FUNCTION_BLOCK FB_AxisAbsolute
VAR	
	// =============== Done signals ============================
	_bResetDone			:BOOL;					// Status of function block MC_Reset
	_bHaltDone			:BOOL;					// Status of function block MC_Halt
	_bStopDone			:BOOL;					// Status of function block MC_Stop
	_bMoveDone			:BOOL;					// Status of function block MC_MoveAbsolute

	// =============== State variables ========================
	_bStatusEnable		:BOOL;					// Enable feedback
	_bStateError		:BOOL;					// Error signal
	_bMoveCommandAborted:BOOL;					// Status of function block MC_MoveAbsolute	
	_nStateErrorID		:UDINT;					// Error ID
	_bStateMoving		:BOOL;					// Status of moving
	_fStateActPos		:LREAL;					// Actual Position
	
	// =============== Position Velocity, override ============
	_fTargetPosition	:LREAL;					// Target Position 
	_fTargetVelocity	:LREAL;					// Target Velocity
	fOverride 			:LREAL := 100.0;		// Override 100%
	
	// =============== Axis Limit =============================
	_fMaxPosition		:LREAL;					//	MAX Target Position 
	_fMinPosition		:LREAL;					//	MIN Target Position 
	_fMaxVelocity		:LREAL;					//	MAX Target Velocity
	_fMinVelocity		:LREAL;					//	MIN Target Velocity
	
	// =============== Trigger function blocks ================
	fbTriggerReset		:R_TRIG;				// Trigger to recognize rising edge of reset input
	fbTriggerHalt		:R_TRIG;				// Trigger to recognize rising edge of halt input
	fbTriggerStop		:R_TRIG;				// Trigger to recognize rising edge of stop input
	fbTriggerMove		:R_TRIG;
	
	// =============== Axis reference =========================
	AxisRef				:AXIS_REF;				// Axis reference (process data plc/nc)
	
	// =============== Motion function blocks =================
	fbMcPower 			:MC_Power;				// FB for enable and override
	fbMcReset 			:MC_Reset;				// FB to reset axis
	fbMcStop 			:MC_Stop;				// FB to stop axis
	fbMcHalt			:MC_Halt;				// FB to halt axis
	fbMcMove			:MC_MoveAbsolute;		// FB to move axis (Absolute movement)
END_VAR

// =========================================================
;
// =========================================================

PROPERTY bStateEnable : BOOL
GET
bStateEnable := _bStatusEnable;
END_GET
END_PROPERTY

PROPERTY bStateError : BOOL
GET
bStateError:=_bStateError;
END_GET
END_PROPERTY

PROPERTY bStateHaltDone : BOOL
GET
bStateHaltDone := _bHaltDone;
END_GET
END_PROPERTY

PROPERTY bStateMoveCommandAborted : BOOL
GET
bStateMoveCommandAborted:=_bMoveCommandAborted;
END_GET
END_PROPERTY

PROPERTY bStateMoveDone : BOOL
GET
bStateMoveDone:=_bMoveDone;
END_GET
END_PROPERTY

PROPERTY bStateMoving : BOOL
GET
bStateMoving:=_bStateMoving;
END_GET
END_PROPERTY

PROPERTY bStateResetDone : BOOL
GET
bStateResetDone := _bResetDone;
END_GET
END_PROPERTY

PROPERTY bStateStopDone : BOOL
GET
bStateStopDone:=_bStopDone;
END_GET
END_PROPERTY

METHOD Enable
VAR_INPUT
	bEnable		: BOOL;
END_VAR
// =========================================================

fbMCPower(	Enable 			:= bEnable, 
			Enable_Positive	:= bEnable, 
			Enable_Negative	:= bEnable, 
			Override		:= fOverride,
			Axis			:= AxisRef,
			Status			=> _bStatusEnable);
			
IF fbMcPower.Error THEN
	_bStateError		:= TRUE;
	_nStateErrorID 		:= fbMcPower.ErrorID;
END_IF

AxisRef.ReadStatus();

_bStateMoving	:= AxisRef.Status.Moving;

_fStateActPos	:= AxisRef.NcToPlc.ActPos;

// =========================================================
END_METHOD

//FB_Init は常に暗黙的に使用可能で、主に初期化に使用されます。
//戻り値は評価されません。特定の結果を得るために、メソッドを明示的に宣言し、
//そのメソッドに標準の初期化コードをもったコードを追加することができます。戻り値を評価できます。
METHOD FB_Init: BOOL
VAR_INPUT
    bInitRetains: BOOL; // TRUE: 保持変数は初期化されます (ウォーム リセット、あるいはコールド リセット)
    bInCopyCode: BOOL;  // TRUE: 後でコードをコピーする (オンライン変更) ために、インスタンスをコピーします。
	

	fMaxPosition	:LREAL;
	fMinPosition	:LREAL;
	fMaxVelocity	:LREAL;
	fMinVelocity	:LREAL;
END_VAR
	_fMaxPosition:=fMaxPosition;
	_fMinPosition:=fMinPosition;
	_fMaxVelocity:=fMaxVelocity;
	_fMinVelocity:=fMinVelocity;
END_METHOD

PROPERTY fStateActPos : LREAL
GET
fStateActPos:=_fStateActPos;
END_GET
END_PROPERTY

PROPERTY fTargetPosition : LREAL
GET
fTargetPosition:=_fTargetPosition;
END_GET
SET
_fTargetPosition:=LIMIT(_fMinPosition,fTargetPosition,_fMaxPosition);
END_SET
END_PROPERTY

PROPERTY fTargetVelocity : LREAL
GET
fTargetVelocity := _fTargetVelocity;
END_GET
SET
_fTargetVelocity :=LIMIT(_fMinVelocity ,fTargetVelocity,_fMaxVelocity);
END_SET
END_PROPERTY

METHOD Halt
VAR_INPUT
	bDriveHalt		: BOOL;					// Request stop
END_VAR
// =========================================================

IF bDriveHalt THEN
	// Move Execute FALSE
	fbMCMove(	Execute	:= FALSE,
				Axis 	:= AxisRef);
ELSE
	// Reset done signal
	_bHaltDone := FALSE;
END_IF

// Trigger
fbTriggerHalt(CLK := bDriveHalt);

IF fbTriggerHalt.Q THEN
	fbMcHalt(	Execute	:= TRUE,
				Axis 	:= AxisRef);
ELSE
	fbMcHalt(Axis := AxisRef);
END_IF

// Done / Error / Command aborted
IF fbMcHalt.Done OR fbMcHalt.Error OR fbMcHalt.CommandAborted THEN
	_bStateError		:= fbMcHalt.Error;
	_nStateErrorID		:= fbMcHalt.ErrorID;
	_bHaltDone 			:= fbMcHalt.Done;
	
	fbMCMove(	Execute	:= FALSE,
				Axis 	:= AxisRef);
				
	fbMcHalt(	Execute	:= FALSE,
				Axis 	:= AxisRef);
END_IF

// =========================================================
END_METHOD

METHOD MoveAbsolute
VAR_INPUT
	bMove		:REFERENCE TO BOOL; 
END_VAR
// =========================================================

IF bMove=TRUE AND(fbMCMove.Error=FALSE OR fbMcHalt.Execute=FALSE OR fbMcStop.Execute=FALSE) THEN
	fbMCMove(	Execute 		:=TRUE,
				Position		:=_fTargetPosition,
				Velocity 		:= _fTargetVelocity,
				Axis 			:= AxisRef,
				Done			=>_bMoveDone,
				CommandAborted	=>_bMoveCommandAborted);	
ELSE
	fbMCMove(	Axis 			:= AxisRef);	
END_IF

// Error / Command aborted
IF fbMCMove.Done OR fbMCMove.Error OR fbMCMove.CommandAborted THEN
	IF fbMcMove.Error THEN
		_bStateError		:= TRUE;
		_nStateErrorID		:= fbMCMove.ErrorID;
	END_IF
	
	bMove:=FALSE;
	
	fbMCMove(	Execute 	:=FALSE,
				Axis 		:= AxisRef);
END_IF

IF fbMcStop.Execute=TRUE OR fbMcHalt.Execute=TRUE THEN
	bMove:=FALSE;
END_IF
END_METHOD

PROPERTY nStateErrorID : UDINT
GET
nStateErrorID:=_nStateErrorID;
END_GET
END_PROPERTY

METHOD Reset
VAR_INPUT
	bDriveReset		: BOOL;					// Request reset
END_VAR
// =========================================================

IF NOT bDriveReset THEN
	_bResetDone 	:= FALSE;
END_IF

// Trigger
fbTriggerReset(CLK := bDriveReset);

IF fbTriggerReset.Q THEN
	_bResetDone		:= FALSE;
	
	fbMcReset(Execute := TRUE, Axis := AxisRef);
ELSE
	fbMcReset(Axis := AxisRef);
END_IF

// Done / Error
IF fbMcReset.Done OR fbMcReset.Error THEN
	_bStateError		:= fbMcReset.Error;
	_nStateErrorID		:= fbMcReset.ErrorID;
	_bResetDone 		:= fbMcReset.Done;

	fbMcReset(	Execute	:= FALSE,
				Axis 	:= AxisRef);
END_IF

// =========================================================
END_METHOD

METHOD Stop
VAR_INPUT
	bDriveStop		: BOOL;					// Request stop
END_VAR
// =========================================================

IF bDriveStop THEN
	// Move Execute FALSE
	fbMCMove(	Execute	:= FALSE,
				Axis 	:= AxisRef);
ELSE
	// Reset done signal
	_bStopDone := FALSE;
END_IF

// Trigger
fbTriggerStop(CLK := bDriveStop);

IF fbTriggerStop.Q THEN
	fbMcStop(	Execute	:= TRUE,
				Axis 	:= AxisRef);
ELSE
	fbMcStop(Axis := AxisRef);
END_IF

// Done / Error / Command aborted
IF fbMcStop.Done OR fbMcStop.Error OR fbMcStop.CommandAborted THEN
	_bStateError		:= fbMcStop.Error;
	_nStateErrorID 		:= fbMcStop.ErrorID;
	_bStopDone 			:= fbMcStop.Done;
	
	fbMCMove(	Execute	:= FALSE,
				Axis 	:= AxisRef);
				
	fbMcStop(	Execute	:= FALSE,
				Axis 	:= AxisRef);
END_IF

// =========================================================
END_METHOD

END_FUNCTION_BLOCK

(* stored: Version 1.1.0.1, ProductVersion 3.1.4026.11
   POU FB_AxisAbsolute: Id {13905c50-061e-47bd-88e1-faf6cd8ad728}, SpecialFunc None
   Property bStateEnable: Id {b623c1c1-f1c5-4202-a065-02024e90e038}
   Get Get: Id {fb4bbe37-ff9a-47af-9c53-30be12f9e058}
   Property bStateError: Id {092893f6-98d3-4487-baa8-93e66efc12a1}
   Get Get: Id {fd3d20a1-36c2-4f32-93ee-18cb01becb8c}
   Property bStateHaltDone: Id {f7de6af1-b5e5-48d8-b512-773820eeee42}
   Get Get: Id {f6a7a426-06e5-4d4b-8c96-62c52d509c00}
   Property bStateMoveCommandAborted: Id {cef249cc-f1c2-4cc8-85c1-541688cd5c69}
   Get Get: Id {a3d32fe0-47e5-4e51-b623-7951d31f69c1}
   Property bStateMoveDone: Id {6198d3a8-ba94-4f92-9011-e865f254b2a2}
   Get Get: Id {b0882baf-0590-4f26-9187-a31096344f10}
   Property bStateMoving: Id {b25fddbe-ad1a-4469-9197-bd51ac3888c0}
   Get Get: Id {79c7942e-f1eb-4237-9662-b5a72f4126a6}
   Property bStateResetDone: Id {51f3a4de-1d38-488f-b402-3183f4c04168}
   Get Get: Id {04c36a28-a9c4-4734-940e-933f64603157}
   Property bStateStopDone: Id {e0b8efe4-3e7d-4b41-8308-d3cbdfb03e2c}
   Get Get: Id {d0fe241d-85d6-47a1-96fc-b3aab94999c5}
   Method Enable: Id {2218bf4b-e6a5-4385-8a61-3d59b9953884}
   Method FB_Init: Id {a51839ba-3519-4ac0-900f-65592382ed92}
   Property fStateActPos: Id {459a73ba-42e1-4b1a-8cdb-74dcaacbbc2f}
   Get Get: Id {4008270e-7e9d-4245-8293-afed7d19d752}
   Property fTargetPosition: Id {77146afd-a1df-4ddb-82da-373341e634e6}
   Get Get: Id {b639191e-3a45-47e0-9665-affaec67bafa}
   Set Set: Id {60b0eb9f-25a0-4f88-8ef9-938c0a2f5a1f}
   Property fTargetVelocity: Id {072eee44-9a89-46ff-9c6c-081e21838b82}
   Get Get: Id {5608d6f9-66c0-4ccb-b31f-4fe6dd87dabd}
   Set Set: Id {70932f21-070c-4a8e-a2f5-0d6642329682}
   Method Halt: Id {e88a2abb-6023-4065-9098-7fa187efe6ad}
   Method MoveAbsolute: Id {16ab69b9-b24d-46b6-acf0-f1ab70404dae}
   Property nStateErrorID: Id {393e9573-61b8-4020-8aeb-991444f3a449}
   Get Get: Id {c1f8ed2c-525f-48c1-8881-05e641af6bd6}
   Method Reset: Id {ea6409fe-eb80-4f4d-b54a-780889e04b6e}
   Method Stop: Id {befb5a74-67aa-4deb-96cf-8551f6226c61} *)
